RoboDK station: Assistive_UR5e _Roc_Maite.rdk

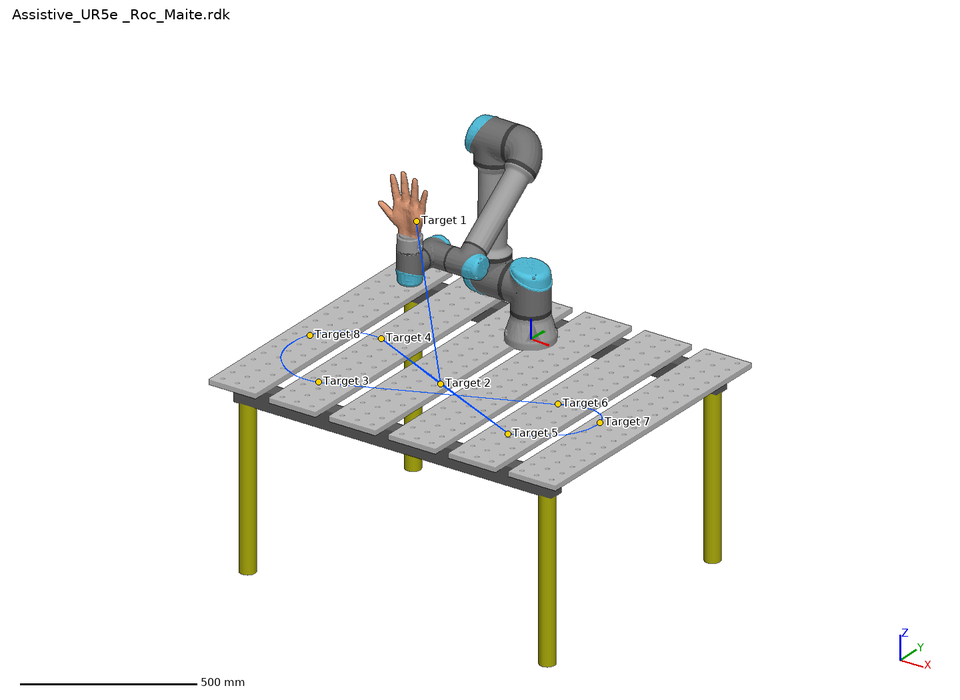
[picture v0: the station drawn from its stored meshes, robots at their saved joint values, targets as dots, program paths as lines]
Station Assistive_UR5e_SW (saved by RoboDK 5.9.2). Poses are relative to the parent item; angles as X-Y-Z fixed-axis rotations.
  - frame UR5e Base at (0, 0, 0) mm, rotated rx 0 ry 0 rz -4.29 deg
    - robot UR5e: 6 axes, payload 5 kg, reach 850 mm, repeatability 0.03 mm, weight 18.4 kg
        modified DH rows (alpha deg, a mm, theta deg, d mm): 0, 0, 0, 162.5; 90, 0, 180, 0; 0, 425, 0, 0; 0, 392.25, 0, 133.3; -90, 0, 0, 99.7; 90, 0, 180, 99.6
        joint limits [-360, -360, -360, -360, -360, -360] to [360, 360, 360, 360, 360, 360]; home [0, -90, -90, 0, 90, 0]; saved at [-86.437, -88.119, -128.455, 306.747, -90.224, 91.317]
      - tool Hand, TCP at (0, 0, 50) mm, size 54.8 x 155.9 x 193.5 mm, geometry from Hand.stl
  - frame World at (0, 0, 0) mm
    - object Table at (0, 0, 0) mm, size 1193.8 x 965.2 x 609.6 mm, geometry from welding_table.sld
    - target Target 1 (Cartesian target) at (-107.58, -407.78, 503.45) mm, rotated rx 0.23 ry 0.17 rz 94.88 deg; joints [-82.143, -88.119, -128.455, 306.747, -90.224, 91.317] of UR5e
    - target Target 2 (Cartesian target) at (5.96, -450.97, 40.88) mm, rotated rx -158.75 ry -89.44 rz -111.81 deg; joints [-58.054, -120.175, -141.349, 260.929, -61.792, 90.485] of UR5e
    - target Target 3 (Cartesian target) at (-285.7, -635.85, 39.45) mm, rotated rx -119.29 ry -89.44 rz -150.46 deg; joints [-102.538, -137.075, -95.636, 232.423, -107.092, 90.406] of UR5e
    - target Target 4 (Cartesian target) at (-298.09, -308.11, 40.77) mm, rotated rx -132.42 ry -89.44 rz -137.57 deg; joints [-124.451, -121.761, -135.373, 256.647, -128.752, 90.111] of UR5e
    - target Target 5 (Cartesian target) at (348.15, -608.2, 42.97) mm, rotated rx -137.88 ry -89.44 rz -133.28 deg; joints [-34.923, -137.867, -92.908, 230.099, -38.066, 90.91] of UR5e
    - target Target 6 (Cartesian target) at (311.66, -310.43, 6.97) mm, rotated rx 91.72 ry -75.42 rz -1.12 deg; joints [-0.686, -128.677, -131.748, 255.929, -5.546, 79.898] of UR5e
    - target Target 7 (Cartesian target) at (519.36, -402.87, 43.66) mm, rotated rx -153.9 ry -89.44 rz -116.1 deg; joints [-8.365, -160.477, -85.824, 63.999, 12.674, -87.506] of UR5e
    - target Target 8 (joint target) at (-477.57, -402.91, 39.36) mm, rotated rx -153.9 ry -89.44 rz -116.1 deg; joints [-133.488, -159.294, -92.115, 70.658, 137.785, -90.309] of UR5e
  - program Init (3 instructions, listed below)
  - program Cleaning_table (13 instructions, listed below)
  - program Give_me_5! (5 instructions, listed below)
  - program MainProgram (4 instructions, listed below)
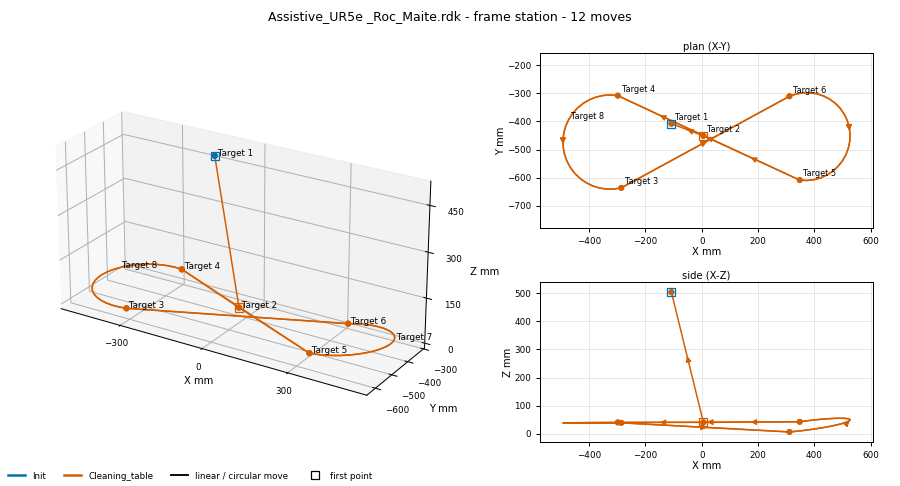
[picture p0: tool path of Assistive_UR5e _Roc_Maite.rdk in frame station, 12 of 15 moves have a stored position in this frame; points joined in program order, loops and branches not executed]

--- program Init (robot UR5e) ---
  Est. Ref.: UR5e Base
  Est. herr: Hand
  MoveJ (Target 1)

--- program Cleaning_table (robot UR5e) ---
  Est. Ref.: UR5e Base
  Est. herr: Hand
  MoveL (Target 2)
  MoveL (Target 4)
  MoveC (Target 8, Target 3)
  MoveL (Target 6)
  MoveC (Target 7, Target 5)
  MoveL (Target 4)
  MoveC (Target 8, Target 3)
  MoveL (Target 6)
  MoveC (Target 7, Target 5)
  MoveL (Target 2)
  MoveL (Target 1)

--- program Give_me_5! (robot UR5e) ---
  Est. Ref.: UR5e Base
  Est. herr: Hand
  MoveL (App_give5) [its target is no longer in the station]
  MoveL (Give5) [its target is no longer in the station]
  MoveL (App_give5) [its target is no longer in the station]

--- program MainProgram (robot UR5e) ---
  Llamar Init
  Llamar Hand_shake
  Llamar Give_me_5!
  Llamar Init
